TYPE ST_MS4208_ETCOut :
STRUCT
	stEFUInputsDevice	AT%I* :	ST_EFU_Device_Inputs;	
	stEFUUs				:	ST_EFU_Data	;
	stEFU_Up1			:	ST_EFU_Data	;
	stEFU_Up2			:	ST_EFU_Data	;
END_STRUCT
END_TYPE

(* stored: Version 1.1.0.1
   DUT ST_MS4208_ETCOut: Id {5fe9215b-ba6c-4fbb-9d61-72db53e88ac4} *)
